// TIA Portal project "Traffic Light" (V16)

(* hardware
DEVICE "S7-1200 station_1"  S7-1200 Station
   slot 0: "Rack_0"  S7-1200 Rack  Rack  V1.0
   slot 1: "PLC_1"  CPU 1212C AC/DC/Rly  6ES7 212-1BE40-0XB0  V4.0
*)

// ===== PLC "PLC_1"  CPU 1212C AC/DC/Rly =====

VAR_GLOBAL   // PLC tag table "Default tag table"
   "start1" AT %I0.2 : Bool;
   "K1 GREEN" AT %Q0.0 : Bool;
   "stop1" AT %I0.4 : Bool;
   "k2 YELLOW" AT %Q0.1 : Bool;
   "T1 tag" AT %M0.0 : Bool;
   "X" AT %M0.2 : Bool;
   "K3 RED" AT %Q0.2 : Bool;
   "STOP" AT %I0.3 : Bool;
END_VAR

// folder: System blocks/Program resources

DATA_BLOCK "TIMER"   // DB1
{ S7_Optimized_Access := 'TRUE' }
AUTHOR : Simatic
FAMILY : IEC
NAME : IEC_TMR
VERSION : 1.0
// stored: InstanceOfName IEC_TIMER
"IEC_TIMER"
BEGIN
END_DATA_BLOCK

// folder: (top level)

ORGANIZATION_BLOCK "Main"   // OB1, LAD, ProgramCycle
TITLE = "Main Program Sweep (Cycle)"
{ S7_Optimized_Access := 'TRUE' }
VERSION : 0.1
   VAR_INPUT
      Initial_Call : Bool;   // Initial call of this OB
      Remanence : Bool;   // =True, if remanent data are available
   END_VAR
BEGIN

REGION Network 1: start
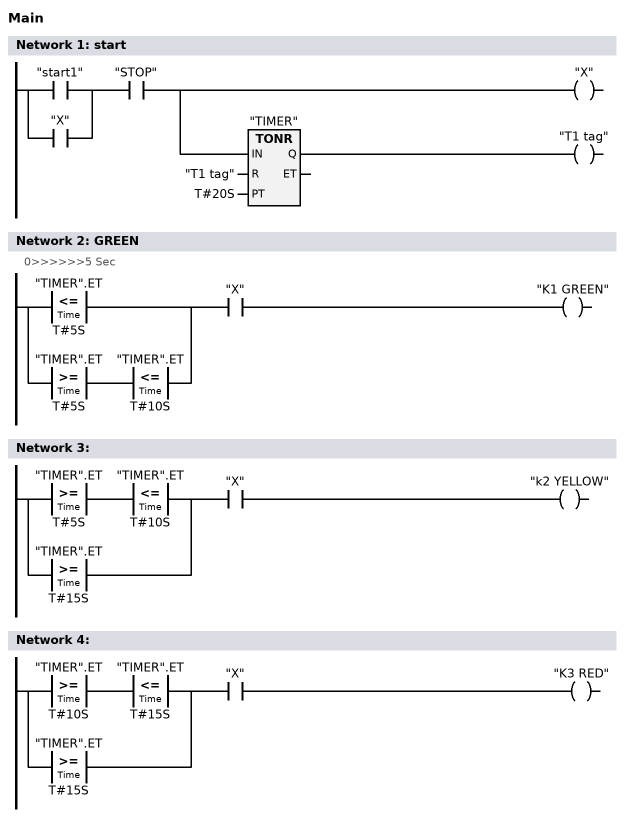
   "X" := ("start1" OR "X") AND "STOP";
   "TIMER".TONR(IN := "X", R := "T1 tag", PT := T#20S);
   "T1 tag" := "TIMER".Q;
END_REGION

REGION Network 2: GREEN
   // 0>>>>>>5 Sec
   RUNG wire#powerrail
      { S7_Templates := "SrcType := Time" } LE_Contact(in1 := "TIMER".ET, in2 := T#5S)
      wire#w1
      Contact( "X" )
      Coil( "K1 GREEN" )
   END_RUNG
   RUNG wire#powerrail
      { S7_Templates := "SrcType := Time" } GE_Contact(in1 := "TIMER".ET, in2 := T#5S)
      { S7_Templates := "SrcType := Time" } LE_Contact(in1 := "TIMER".ET, in2 := T#10S)
   END_RUNG wire#w1
   // the same network as SCL:
   "K1 GREEN" := (("TIMER".ET <= T#5S) OR (("TIMER".ET >= T#5S) AND ("TIMER".ET <= T#10S))) AND "X";
END_REGION

REGION Network 3
   RUNG wire#powerrail
      { S7_Templates := "SrcType := Time" } GE_Contact(in1 := "TIMER".ET, in2 := T#5S)
      { S7_Templates := "SrcType := Time" } LE_Contact(in1 := "TIMER".ET, in2 := T#10S)
      wire#w1
      Contact( "X" )
      Coil( "k2 YELLOW" )
   END_RUNG
   RUNG wire#powerrail
      { S7_Templates := "SrcType := Time" } GE_Contact(in1 := "TIMER".ET, in2 := T#15S)
   END_RUNG wire#w1
   // the same network as SCL:
   "k2 YELLOW" := ((("TIMER".ET >= T#5S) AND ("TIMER".ET <= T#10S)) OR ("TIMER".ET >= T#15S)) AND "X";
END_REGION

REGION Network 4
   RUNG wire#powerrail
      { S7_Templates := "SrcType := Time" } GE_Contact(in1 := "TIMER".ET, in2 := T#10S)
      { S7_Templates := "SrcType := Time" } LE_Contact(in1 := "TIMER".ET, in2 := T#15S)
      wire#w1
      Contact( "X" )
      Coil( "K3 RED" )
   END_RUNG
   RUNG wire#powerrail
      { S7_Templates := "SrcType := Time" } GE_Contact(in1 := "TIMER".ET, in2 := T#15S)
   END_RUNG wire#w1
   // the same network as SCL:
   "K3 RED" := ((("TIMER".ET >= T#10S) AND ("TIMER".ET <= T#15S)) OR ("TIMER".ET >= T#15S)) AND "X";
END_REGION
END_ORGANIZATION_BLOCK